// instrument joints control
FUNCTION_BLOCK FB_BasicInstruControlNew
VAR_INPUT
END_VAR
VAR_OUTPUT
END_VAR
VAR
	// instrument PID control paramters
	m_instruKp:ARRAY[1..5] OF LREAL:=[5(3)];
	m_instruKd:ARRAY[1..5] OF LREAL:=[5(0.04)];
	m_instruKi:ARRAY[1..5] OF LREAL:=[5(10.0)];
	m_instruKiLimit:ARRAY[1..5] OF LREAL:=[5(150.0)];
	m_instruCtrlLimit:ARRAY[1..5] OF LREAL:=[2(300.0), 3(700.0)];
	
	// gripper force level threshold for variable PID parameter
	m_forceLevelThres : ARRAY[1..3] OF LREAL := [40, 70, 101];
	
	// yaw PID control (when fingers grasp with force)
	m_yawKp:ARRAY[1..3] OF LREAL:=[2, 2, 2];
	m_yawKd:ARRAY[1..3] OF LREAL:=[0.025, 0.025, 0.025];
	m_yawKi:ARRAY[1..3] OF LREAL:=[10, 15, 20];
	m_yawKiLimit:LREAL:=300.0;
	m_yawCtrlLimit:LREAL:=700.0;
	
	// max grip force/current(mA)
	m_maxGripForce:LREAL;
	m_maxGripCurrent:LREAL:=300.0;
	
	// max gripper finger control force/current(mA)
	m_maxGripCtrlForce:LREAL;
	m_maxGripCtrlCurrent:LREAL:=600.0;
	
	// PID for instrument joint position
	m_instruJntCtrl:ARRAY[1..5] OF FB_PID;

	// PID for instrument yaw angle 
	m_instruYawCtrl : FB_PID;
	
	// command instrument joint position and velocity
	m_instruCmdJntPos:Vec5d;
	m_instruCmdJntVel:Vec5d;
	
	// current instrument joint position and velocity
	m_instruCurJntPos: Vec5d;
	m_instruCurJntVel:Vec5d;
	
	// grasp force level
	m_graspForceLevel:Lreal :=0;
	
	// instrument joint control torque(when gripper is open)
	m_instruJntCtrlTrq:Vec5d:=[5(0.0)];

	// instrument yaw control torque(when gripper is closed)
	m_instruYawCtrlTrq:LREAL;
		
	// current gripper yaw velocity
	m_instruCurYawVel:LREAL;
	
	// yaw angle error(deg)
	m_yawAngErr : LREAL;
	
	// backlash compensation variables
	m_jntBacklash:ARRAY[1..5] OF LREAL:=[5(0)];
	m_instruLastCmdJntPos:Vec5d;
	
	//pitch back lash on account of  Yaw
	m_pitchBackLash : ARRAY [1..5] OF LREAL := [5(0)];
	m_pitchBackLashLpf :FB_LowPassFilter;
	
	// grip yaw compensation variables
 	m_gripYawCompAng :LREAL;
 	m_maxGripYawCompAng :LREAL;
	m_lastCmdYawAng:LREAL;
	m_jntMoveStep:LREAL := 0.5*g_deg2Rad;
	
	m_maxPitchCompAngle : LREAL := 5*g_deg2Rad;
	
	// filter cut-off frequency for pitch back lash
	m_cmdJntPosLpfCutoffFreq : LREAL :=3;
END_VAR

METHOD calcBacklash : BOOL
VAR_IN_OUT CONSTANT
	// instrument joint command position
	i_cmdInstruJntPos :Vec5d;
	
	// command yaw position
	i_cmdYawPos : LREAL;
	
	// slave arm data
	i_slaveArm :FB_SlaveArm;
END_VAR

VAR
	i:INT;
	deltaAng:LREAL;
	pitchBackLash : LREAL;
END_VAR
// backslash compensation
FOR i:=1 TO 4 DO
	// integral compensated backslash angle
	deltaAng:=i_cmdInstruJntPos[i]-m_instruLastCmdJntPos[i];
	IF ABS(deltaAng)>m_jntMoveStep THEN
		m_jntBacklash [i] := m_jntBacklash [i] + m_jntMoveStep*sign(deltaAng);
		m_instruLastCmdJntPos[i] := i_cmdInstruJntPos[i];
	END_IF
END_FOR


// exert grip force 
IF m_graspForceLevel >0  THEN
	
	// clear grip finger backlash
	m_jntBacklash [1]:=0;
	m_jntBacklash [2]:=0;
	
	// determin max compensated angle based on grip force 
	FOR i:=1 TO 4 DO 
		IF m_graspForceLevel<= g_instruGripYawCompForceLevel[i] THEN
			m_maxGripYawCompAng := g_instruGripYawCompAng[i];
			EXIT;
		END_IF
	END_FOR

	// compensate yaw joint angle in case it's driven by force difference between two fingers
	pitchBackLash := ((i_slaveArm.filtJntCurrent[5] - i_slaveArm.filtJntCurrent[4])/m_maxGripCtrlCurrent)*m_maxPitchCompAngle;
	m_pitchBackLash[3] := m_pitchBackLashLpf.run(i_rawData:=pitchBackLash );
	
	// determin  compensated angle
	IF ABS(i_cmdYawPos - m_lastCmdYawAng) > m_jntMoveStep  THEN
		// determin  compensated yaw  angle
		IF (i_cmdYawPos - m_lastCmdYawAng) * m_gripYawCompAng <= 0 THEN
			m_gripYawCompAng := m_gripYawCompAng + 0.5*m_jntMoveStep * sign(i_cmdYawPos-m_lastCmdYawAng);
		ELSE
			m_gripYawCompAng := m_gripYawCompAng + 0.5*m_jntMoveStep * sign(i_cmdYawPos-m_lastCmdYawAng);
		END_IF
		m_lastCmdYawAng := i_cmdYawPos;
	END_IF
	m_gripYawCompAng := LIMIT(-m_maxGripYawCompAng, m_gripYawCompAng,m_maxGripYawCompAng);
	

ELSE
	m_pitchBackLash[3] := 0;
	m_gripYawCompAng:=0;
	m_lastCmdYawAng := i_cmdYawPos;
END_IF

// limit compensated backslash angle
FOR i:=1 TO 4 DO

	IF i<3 THEN 
		IF g_instruBacklashDir[i] > 0 THEN
			m_jntBacklash [i] := LIMIT(0, m_jntBacklash[i], i_slaveArm.instrument.instruTypeInfo.m_instruYawBacklash);		
		ELSE
			m_jntBacklash [i] := LIMIT(-i_slaveArm.instrument.instruTypeInfo.m_instruYawBacklash, m_jntBacklash[i], 0);	
		END_IF

	ELSIF i=3 THEN
		IF g_instruBacklashDir[i] > 0 THEN
			m_jntBacklash [i] := LIMIT(0, m_jntBacklash[i], i_slaveArm.instrument.instruTypeInfo.m_instruPitchBachlash);
		ELSE
			m_jntBacklash [i] := LIMIT(-i_slaveArm.instrument.instruTypeInfo.m_instruPitchBachlash, m_jntBacklash[i], 0);	
		END_IF
	ELSE
		m_jntBacklash [i]:=0;
	END_IF
	
END_FOR
END_METHOD

METHOD init : BOOL
VAR_IN_OUT CONSTANT
	i_slaveArm:FB_SlaveArm;
END_VAR

VAR
	i,j:INT;
	currentRatioMotor2Jnt:LREAL;
END_VAR
m_graspForceLevel:=0;

// init controller
currentRatioMotor2Jnt:=GVL_SlaveMotorParameters.g_motorTrqConstArm4[4]*GVL_SlaveMotorParameters.g_motorReductionArm4[4]/1000;
m_maxGripForce := m_maxGripCurrent * currentRatioMotor2Jnt;
m_maxGripCtrlForce := m_maxGripCtrlCurrent * currentRatioMotor2Jnt;
FOR i:=1 TO 4 DO
	m_jntBacklash[i] := 0;
	m_instruCmdJntPos[i]:=i_slaveArm.curJntPos[i+3];
	
	m_instruCmdJntVel[i]:=0;
	
	m_instruJntCtrl[i].init(g_slaveArmCtrlCycleTime,m_instruKp[i],m_instruKd[i],m_instruKi[i],
		m_instruKiLimit[i]* currentRatioMotor2Jnt,	m_instruCtrlLimit[i]*currentRatioMotor2Jnt);
	
	m_instruLastCmdJntPos[i]:=m_instruCmdJntPos[i];
END_FOR
m_instruYawCtrl.init(g_slaveArmCtrlCycleTime,m_yawKp[1],m_yawKd[1],m_yawKi[1],m_yawKiLimit*currentRatioMotor2Jnt, m_yawCtrlLimit*currentRatioMotor2Jnt);
m_pitchBackLashLpf.init(1, m_cmdJntPosLpfCutoffFreq, g_slaveArmCtrlFreq);
END_METHOD

METHOD run : BOOL
VAR_IN_OUT CONSTANT
	// instrument joint command position
	i_cmdInstruJntPos :Vec5d;
	
	// instrument joint command velocity
	i_cmdInstruJntVel :Vec5d;
	
	// command yaw position
	i_cmdYawPos : LREAL;
	
	// command yaw velocity
	i_cmdYawVel :LREAL;
	
	// command grip force level
	i_cmdGripForceLevel:LREAL;
	
	// slave arm data
	i_slaveArm :FB_SlaveArm;
END_VAR

VAR_OUTPUT
	// joint control torque
	o_cmdJntTrq:Vec5d;
END_VAR

VAR
	i: INT;
	deltaAng:LREAL;
END_VAR
m_graspForceLevel:=LIMIT(0,i_cmdGripForceLevel ,  100)	;

// calculate instrument backlash
calcBacklash(i_cmdInstruJntPos, i_cmdYawPos, i_slaveArm);


// joint position control
FOR i:=1 TO 4 DO	
	m_instruCmdJntPos[i]:=i_cmdInstruJntPos[i];
	m_instruCmdJntVel[i]:=i_cmdInstruJntVel[i];
	m_instruCurJntPos[i]:=i_slaveArm.curJntPos[i+3];
	m_instruCurJntVel[i]:= i_slaveArm.curJntVel[i+3];
	m_instruJntCtrlTrq[i]:=m_instruJntCtrl[i].run(m_instruCmdJntPos[i] + m_jntBacklash[i] + m_pitchBackLash[i] ,m_instruCurJntPos[i], m_instruCmdJntVel[i], m_instruCurJntVel[i]);
END_FOR

m_instruJntCtrlTrq[5]:=0;

m_instruCurYawVel :=i_slaveArm.curDHJntVel[6];
m_yawAngErr:=g_rad2Deg*(i_cmdYawPos-i_slaveArm.curDHJntPos[6]);


// exert grip force 
IF m_graspForceLevel >0  THEN
	
	// varialbe PID control based on different gripper force level
	FOR i:=1 TO 3 DO 
		IF m_graspForceLevel < m_forceLevelThres[i] THEN
			m_instruYawCtrl.setPIDParam(m_yawKp[i],m_yawKd[i],m_yawKi[i]);
			EXIT;
		END_IF
	END_FOR

	// yaw control
	m_instruYawCtrlTrq:=m_instruYawCtrl.run(i_cmdYawPos+m_gripYawCompAng,i_slaveArm.curDHJntPos[6],i_cmdYawVel, m_instruCurYawVel);

	// add feed forward grasp force
	m_instruJntCtrlTrq[1]:= m_maxGripForce*m_graspForceLevel/100.0 + m_instruYawCtrlTrq;
	m_instruJntCtrlTrq[2]:= m_maxGripForce*m_graspForceLevel/100.0 - m_instruYawCtrlTrq;
	m_instruJntCtrlTrq[1]:=LIMIT(-m_maxGripCtrlForce/2.0,m_instruJntCtrlTrq[1], m_maxGripCtrlForce);
	m_instruJntCtrlTrq[2]:=LIMIT(-m_maxGripCtrlForce/2.0,m_instruJntCtrlTrq[2], m_maxGripCtrlForce);
END_IF


o_cmdJntTrq := m_instruJntCtrlTrq;
END_METHOD

END_FUNCTION_BLOCK

(* stored: Version 1.1.0.1, ProductVersion 3.1.4024.11
   POU FB_BasicInstruControlNew: Id {2cc54694-5109-4339-b599-ede4b8dcd0f6}, SpecialFunc None
   Method calcBacklash: Id {aeb9718b-c6f1-4086-a1bf-d28986f24f69}
   Method init: Id {65c72158-b7f0-4f81-9e17-42eb8752ec5c}
   Method run: Id {91885246-8ac4-4aa6-9fed-10291849b120} *)
